Staubli VAL3: programList.pgx

program programList(string& x_sEvent[])
  local num nSize
  local string sEvent
  local num lKey
  local num i
  local string message
begin
  //
  // USE this procedure to view Prog
  // that you have already saved
  //
  cls()
  call use:setView(false)
  //
  // Prog
  //
  call use:listcreate("PROG ")
  // set the path to prog pallet
  //
  call prog:getSize(nSize)
  // refresh the list
  for i=0 to nSize-1
    call prog:get(sEvent,i)
    if sEvent!=""
      call use:listadd(sEvent)
    endIf
  endFor
  call use:listupdate(0)
  call language:message(message,60)
  call use:typeLen(0,13,message,40)
  call language:message(message,-19)
  message=" F7: "+message
  call use:type(0,9,message)
  do
    lKey=get()
    call use:listevent(lKey,i,x_sEvent)
  until lKey==270 or lKey==255 or lKey==277
  if lKey==277
    x_sEvent=""
  endIf
end
